// Image Filtering
NodeFactory.AddNodeAsPrototype('Vision/Image Filtering/F_VN_BilateralFilter', node_F_VN_BilateralFilter);
NodeFactory.AddNodeAsPrototype('Vision/Image Filtering/F_VN_BilateralFilterExp', node_F_VN_BilateralFilterExp);
NodeFactory.AddNodeAsPrototype('Vision/Image Filtering/F_VN_BoxFilter', node_F_VN_BoxFilter);
NodeFactory.AddNodeAsPrototype('Vision/Image Filtering/F_VN_BoxFilterExp', node_F_VN_BoxFilterExp);
NodeFactory.AddNodeAsPrototype('Vision/Image Filtering/F_VN_BrightBorderObjects', node_F_VN_BrightBorderObjects);
NodeFactory.AddNodeAsPrototype('Vision/Image Filtering/F_VN_CreateStructuringElement', node_F_VN_CreateStructuringElement);
//NodeFactory.AddNodeAsPrototype('Vision/Image Filtering/F_VN_CustomFilter', node_F_VN_CustomFilter);
//NodeFactory.AddNodeAsPrototype('Vision/Image Filtering/F_VN_CustomFilterExp', node_F_VN_CustomFilterExp);
NodeFactory.AddNodeAsPrototype('Vision/Image Filtering/F_VN_DarkBorderObjects', node_F_VN_DarkBorderObjects);
NodeFactory.AddNodeAsPrototype('Vision/Image Filtering/F_VN_FillHoles', node_F_VN_FillHoles);
NodeFactory.AddNodeAsPrototype('Vision/Image Filtering/F_VN_GaussianFilter', node_F_VN_GaussianFilter);
NodeFactory.AddNodeAsPrototype('Vision/Image Filtering/F_VN_GaussianFilterExp', node_F_VN_GaussianFilterExp);
NodeFactory.AddNodeAsPrototype('Vision/Image Filtering/F_VN_LaplacianFilter', node_F_VN_LaplacianFilter);
NodeFactory.AddNodeAsPrototype('Vision/Image Filtering/F_VN_LaplacianFilterExp', node_F_VN_LaplacianFilterExp);
NodeFactory.AddNodeAsPrototype('Vision/Image Filtering/F_VN_LocalMaxima', node_F_VN_LocalMaxima);
NodeFactory.AddNodeAsPrototype('Vision/Image Filtering/F_VN_LocalMinima', node_F_VN_LocalMinima);
NodeFactory.AddNodeAsPrototype('Vision/Image Filtering/F_VN_MedianFilter', node_F_VN_MedianFilter);
NodeFactory.AddNodeAsPrototype('Vision/Image Filtering/F_VN_MorphologicalOperator', node_F_VN_MorphologicalOperator);
NodeFactory.AddNodeAsPrototype('Vision/Image Filtering/F_VN_RemoveLocalMaxima', node_F_VN_RemoveLocalMaxima);
NodeFactory.AddNodeAsPrototype('Vision/Image Filtering/F_VN_RemoveLocalMinima', node_F_VN_RemoveLocalMinima);
NodeFactory.AddNodeAsPrototype('Vision/Image Filtering/F_VN_ScharrFilter', node_F_VN_ScharrFilter);
NodeFactory.AddNodeAsPrototype('Vision/Image Filtering/F_VN_ScharrFilterExp', node_F_VN_ScharrFilterExp);
//NodeFactory.AddNodeAsPrototype('Vision/Image Filtering/F_VN_SeparableCustomFilter', node_F_VN_SeparableCustomFilter);
//NodeFactory.AddNodeAsPrototype('Vision/Image Filtering/F_VN_SeparableCustomFilterExp', node_F_VN_SeparableCustomFilterExp);
NodeFactory.AddNodeAsPrototype('Vision/Image Filtering/F_VN_SobelFilter', node_F_VN_SobelFilter);
NodeFactory.AddNodeAsPrototype('Vision/Image Filtering/F_VN_SobelFilterExp', node_F_VN_SobelFilterExp);
NodeFactory.AddNodeAsPrototype('Vision/Image Filtering/F_VN_VarianceFilter', node_F_VN_VarianceFilter);
NodeFactory.AddNodeAsPrototype('Vision/Image Filtering/F_VN_VarianceFilterExp', node_F_VN_VarianceFilterExp);
    
// Image Segmentation
NodeFactory.AddNodeAsPrototype('Vision/Image Segmentation/F_VN_AdaptiveThreshold', node_F_VN_AdaptiveThreshold);
NodeFactory.AddNodeAsPrototype('Vision/Image Segmentation/F_VN_AdaptiveThresholdExp', node_F_VN_AdaptiveThresholdExp);
NodeFactory.AddNodeAsPrototype('Vision/Image Segmentation/F_VN_CheckColorRange', node_F_VN_CheckColorRange);
NodeFactory.AddNodeAsPrototype('Vision/Image Segmentation/F_VN_DoubleThreshold', node_F_VN_DoubleThreshold);
NodeFactory.AddNodeAsPrototype('Vision/Image Segmentation/F_VN_Threshold', node_F_VN_Threshold);
NodeFactory.AddNodeAsPrototype('Vision/Image Segmentation/F_VN_WatershedSegmentationExp', node_F_VN_WatershedSegmentationExp);
NodeFactory.AddNodeAsPrototype('Vision/Image Segmentation/F_VN_SauvolaThreshold', node_F_VN_SauvolaThreshold);

// Keypoint Features
NodeFactory.AddNodeAsPrototype('Vision/Keypoint Features/F_VN_FilterGoodMatches', node_F_VN_FilterGoodMatches);
NodeFactory.AddNodeAsPrototype('Vision/Keypoint Features/F_VN_FindReferenceKeyPointsInImage', node_F_VN_FindReferenceKeyPointsInImage);
NodeFactory.AddNodeAsPrototype('Vision/Keypoint Features/F_VN_FindReferenceKeyPointsInImageAKAZE', node_F_VN_FindReferenceKeyPointsInImageAKAZE);
NodeFactory.AddNodeAsPrototype('Vision/Keypoint Features/F_VN_FindReferenceKeyPointsInImageAKAZEExp', node_F_VN_FindReferenceKeyPointsInImageAKAZEExp);
NodeFactory.AddNodeAsPrototype('Vision/Keypoint Features/F_VN_FindReferenceKeyPointsInImageBRISK', node_F_VN_FindReferenceKeyPointsInImageBRISK);
NodeFactory.AddNodeAsPrototype('Vision/Keypoint Features/F_VN_FindReferenceKeyPointsInImageBRISKExp', node_F_VN_FindReferenceKeyPointsInImageBRISKExp);
NodeFactory.AddNodeAsPrototype('Vision/Keypoint Features/F_VN_FindReferenceKeyPointsInImageExp', node_F_VN_FindReferenceKeyPointsInImageExp);
NodeFactory.AddNodeAsPrototype('Vision/Keypoint Features/F_VN_FindReferenceKeyPointsInImageORB', node_F_VN_FindReferenceKeyPointsInImageORB);
NodeFactory.AddNodeAsPrototype('Vision/Keypoint Features/F_VN_FindReferenceKeyPointsInImageORBExp', node_F_VN_FindReferenceKeyPointsInImageORBExp);
NodeFactory.AddNodeAsPrototype('Vision/Keypoint Features/F_VN_GetMatchCoordinates', node_F_VN_GetMatchCoordinates);
NodeFactory.AddNodeAsPrototype('Vision/Keypoint Features/F_VN_KeyPointsAGAST', node_F_VN_KeyPointsAGAST);
NodeFactory.AddNodeAsPrototype('Vision/Keypoint Features/F_VN_KeyPointsAGASTExp', node_F_VN_KeyPointsAGASTExp);
NodeFactory.AddNodeAsPrototype('Vision/Keypoint Features/F_VN_KeyPointsAndDescriptorsAKAZE', node_F_VN_KeyPointsAndDescriptorsAKAZE);
NodeFactory.AddNodeAsPrototype('Vision/Keypoint Features/F_VN_KeyPointsAndDescriptorsAKAZEExp', node_F_VN_KeyPointsAndDescriptorsAKAZEExp);
NodeFactory.AddNodeAsPrototype('Vision/Keypoint Features/F_VN_KeyPointsAndDescriptorsBRISK', node_F_VN_KeyPointsAndDescriptorsBRISK);
NodeFactory.AddNodeAsPrototype('Vision/Keypoint Features/F_VN_KeyPointsAndDescriptorsBRISKExp', node_F_VN_KeyPointsAndDescriptorsBRISKExp);
NodeFactory.AddNodeAsPrototype('Vision/Keypoint Features/F_VN_KeyPointsAndDescriptorsKAZE', node_F_VN_KeyPointsAndDescriptorsKAZE);
NodeFactory.AddNodeAsPrototype('Vision/Keypoint Features/F_VN_KeyPointsAndDescriptorsKAZEExp', node_F_VN_KeyPointsAndDescriptorsKAZEExp);
NodeFactory.AddNodeAsPrototype('Vision/Keypoint Features/F_VN_KeyPointsAndDescriptorsORB', node_F_VN_KeyPointsAndDescriptorsORB);
NodeFactory.AddNodeAsPrototype('Vision/Keypoint Features/F_VN_KeyPointsAndDescriptorsORBExp', node_F_VN_KeyPointsAndDescriptorsORBExp);
NodeFactory.AddNodeAsPrototype('Vision/Keypoint Features/F_VN_KeyPointsFAST', node_F_VN_KeyPointsFAST);
NodeFactory.AddNodeAsPrototype('Vision/Keypoint Features/F_VN_KeyPointsFASTExp', node_F_VN_KeyPointsFASTExp);
NodeFactory.AddNodeAsPrototype('Vision/Keypoint Features/F_VN_KeyPointsGFTT', node_F_VN_KeyPointsGFTT);
NodeFactory.AddNodeAsPrototype('Vision/Keypoint Features/F_VN_KeyPointsGFTTExp', node_F_VN_KeyPointsGFTTExp);
NodeFactory.AddNodeAsPrototype('Vision/Keypoint Features/F_VN_KeyPointsMSER', node_F_VN_KeyPointsMSER);
NodeFactory.AddNodeAsPrototype('Vision/Keypoint Features/F_VN_KeyPointsMSERExp', node_F_VN_KeyPointsMSERExp);
NodeFactory.AddNodeAsPrototype('Vision/Keypoint Features/F_VN_KeyPointsSB', node_F_VN_KeyPointsSB);
NodeFactory.AddNodeAsPrototype('Vision/Keypoint Features/F_VN_KeyPointsSBExp', node_F_VN_KeyPointsSBExp);
NodeFactory.AddNodeAsPrototype('Vision/Keypoint Features/F_VN_MatchDescriptorsBF', node_F_VN_MatchDescriptorsBF);
NodeFactory.AddNodeAsPrototype('Vision/Keypoint Features/F_VN_MatchDescriptorsBFExp', node_F_VN_MatchDescriptorsBFExp);
NodeFactory.AddNodeAsPrototype('Vision/Keypoint Features/F_VN_MatchDescriptorsFlannLsh', node_F_VN_MatchDescriptorsFlannLsh);
NodeFactory.AddNodeAsPrototype('Vision/Keypoint Features/F_VN_MatchDescriptorsFlannLshExp', node_F_VN_MatchDescriptorsFlannLshExp);
NodeFactory.AddNodeAsPrototype('Vision/Keypoint Features/F_VN_MatchDescriptorsKnnBF', node_F_VN_MatchDescriptorsKnnBF);
NodeFactory.AddNodeAsPrototype('Vision/Keypoint Features/F_VN_MatchDescriptorsKnnBFExp', node_F_VN_MatchDescriptorsKnnBFExp);
NodeFactory.AddNodeAsPrototype('Vision/Keypoint Features/F_VN_MatchDescriptorsKnnFlannLsh', node_F_VN_MatchDescriptorsKnnFlannLsh);
NodeFactory.AddNodeAsPrototype('Vision/Keypoint Features/F_VN_MatchDescriptorsKnnFlannLshExp', node_F_VN_MatchDescriptorsKnnFlannLshExp);
NodeFactory.AddNodeAsPrototype('Vision/Keypoint Features/F_VN_RegionsMSER', node_F_VN_RegionsMSER);
NodeFactory.AddNodeAsPrototype('Vision/Keypoint Features/F_VN_RegionsMSERExp', node_F_VN_RegionsMSERExp);

// Machine Learning
//NodeFactory.AddNodeAsPrototype('Vision/Machine Learning/F_VN_CreateBoostClassifier', node_F_VN_CreateBoostClassifier);
//NodeFactory.AddNodeAsPrototype('Vision/Machine Learning/F_VN_CreateBoostClassifierExp', node_F_VN_CreateBoostClassifierExp);
//NodeFactory.AddNodeAsPrototype('Vision/Machine Learning/F_VN_CreateBoostClassifierExp2', node_F_VN_CreateBoostClassifierExp2);
//NodeFactory.AddNodeAsPrototype('Vision/Machine Learning/F_VN_CreateKmppModel', node_F_VN_CreateKmppModel);
//NodeFactory.AddNodeAsPrototype('Vision/Machine Learning/F_VN_CreateKmppModelExp', node_F_VN_CreateKmppModelExp);
//NodeFactory.AddNodeAsPrototype('Vision/Machine Learning/F_VN_CreateKnnModel', node_F_VN_CreateKnnModel);
//NodeFactory.AddNodeAsPrototype('Vision/Machine Learning/F_VN_CreateLbgModel', node_F_VN_CreateLbgModel);
//NodeFactory.AddNodeAsPrototype('Vision/Machine Learning/F_VN_CreateLbgModelExp', node_F_VN_CreateLbgModelExp);
//NodeFactory.AddNodeAsPrototype('Vision/Machine Learning/F_VN_CreateLdaTransform', node_F_VN_CreateLdaTransform);
//NodeFactory.AddNodeAsPrototype('Vision/Machine Learning/F_VN_CreateLdaTransformViaComponentNum', node_F_VN_CreateLdaTransformViaComponentNum);
//NodeFactory.AddNodeAsPrototype('Vision/Machine Learning/F_VN_CreateNbcModel', node_F_VN_CreateNbcModel);
//NodeFactory.AddNodeAsPrototype('Vision/Machine Learning/F_VN_CreatePcaTransform', node_F_VN_CreatePcaTransform);
//NodeFactory.AddNodeAsPrototype('Vision/Machine Learning/F_VN_CreatePcaTransformViaComponentNum', node_F_VN_CreatePcaTransformViaComponentNum);
//NodeFactory.AddNodeAsPrototype('Vision/Machine Learning/F_VN_CreatePcaTransformViaVariance', node_F_VN_CreatePcaTransformViaVariance);
//NodeFactory.AddNodeAsPrototype('Vision/Machine Learning/F_VN_CreateRTreesModel', node_F_VN_CreateRTreesModel);
//NodeFactory.AddNodeAsPrototype('Vision/Machine Learning/F_VN_CreateRTreesModelExp', node_F_VN_CreateRTreesModelExp);
//NodeFactory.AddNodeAsPrototype('Vision/Machine Learning/F_VN_CreateRTreesModelExp2', node_F_VN_CreateRTreesModelExp2);
//NodeFactory.AddNodeAsPrototype('Vision/Machine Learning/F_VN_CreateStaModel', node_F_VN_CreateStaModel);
//NodeFactory.AddNodeAsPrototype('Vision/Machine Learning/F_VN_CreateStaModelExp', node_F_VN_CreateStaModelExp);
//NodeFactory.AddNodeAsPrototype('Vision/Machine Learning/F_VN_CreateStaModelExp2', node_F_VN_CreateStaModelExp2);
//NodeFactory.AddNodeAsPrototype('Vision/Machine Learning/F_VN_CreateSvmModel', node_F_VN_CreateSvmModel);
//NodeFactory.AddNodeAsPrototype('Vision/Machine Learning/F_VN_CreateSvmModelExp', node_F_VN_CreateSvmModelExp);
//NodeFactory.AddNodeAsPrototype('Vision/Machine Learning/F_VN_CreateSvmModelExp2', node_F_VN_CreateSvmModelExp2);
//NodeFactory.AddNodeAsPrototype('Vision/Machine Learning/F_VN_CreateSvmSgdClassifier', node_F_VN_CreateSvmSgdClassifier);
//NodeFactory.AddNodeAsPrototype('Vision/Machine Learning/F_VN_CreateSvmSgdClassifierExp', node_F_VN_CreateSvmSgdClassifierExp);
//NodeFactory.AddNodeAsPrototype('Vision/Machine Learning/F_VN_FeatureScaling', node_F_VN_FeatureScaling);
//NodeFactory.AddNodeAsPrototype('Vision/Machine Learning/F_VN_FeatureScalingExp', node_F_VN_FeatureScalingExp);
//NodeFactory.AddNodeAsPrototype('Vision/Machine Learning/F_VN_FeatureTransform', node_F_VN_FeatureTransform);
//NodeFactory.AddNodeAsPrototype('Vision/Machine Learning/F_VN_GetBatchClusters', node_F_VN_GetBatchClusters);
//NodeFactory.AddNodeAsPrototype('Vision/Machine Learning/F_VN_GetBatchClustersExp', node_F_VN_GetBatchClustersExp);
//NodeFactory.AddNodeAsPrototype('Vision/Machine Learning/F_VN_GetBatchNovelties', node_F_VN_GetBatchNovelties);
//NodeFactory.AddNodeAsPrototype('Vision/Machine Learning/F_VN_GetClusterCenter', node_F_VN_GetClusterCenter);
//NodeFactory.AddNodeAsPrototype('Vision/Machine Learning/F_VN_GetClusterNum', node_F_VN_GetClusterNum);
//NodeFactory.AddNodeAsPrototype('Vision/Machine Learning/F_VN_GetFeatureScales', node_F_VN_GetFeatureScales);
//NodeFactory.AddNodeAsPrototype('Vision/Machine Learning/F_VN_GetSampleCluster', node_F_VN_GetSampleCluster);
//NodeFactory.AddNodeAsPrototype('Vision/Machine Learning/F_VN_GetSampleClusterExp', node_F_VN_GetSampleClusterExp);
//NodeFactory.AddNodeAsPrototype('Vision/Machine Learning/F_VN_GetSampleNovelty', node_F_VN_GetSampleNovelty);
//NodeFactory.AddNodeAsPrototype('Vision/Machine Learning/F_VN_InverseFeatureScaling', node_F_VN_InverseFeatureScaling);
//NodeFactory.AddNodeAsPrototype('Vision/Machine Learning/F_VN_InverseFeatureScaling_REAL', node_F_VN_InverseFeatureScaling_REAL);
//NodeFactory.AddNodeAsPrototype('Vision/Machine Learning/F_VN_InverseFeatureScalingExp', node_F_VN_InverseFeatureScalingExp);
//NodeFactory.AddNodeAsPrototype('Vision/Machine Learning/F_VN_InverseFeatureScalingExp_REAL', node_F_VN_InverseFeatureScalingExp_REAL);
//NodeFactory.AddNodeAsPrototype('Vision/Machine Learning/F_VN_InverseFeatureTransform', node_F_VN_InverseFeatureTransform);
//NodeFactory.AddNodeAsPrototype('Vision/Machine Learning/F_VN_PredictBatch', node_F_VN_PredictBatch);
//NodeFactory.AddNodeAsPrototype('Vision/Machine Learning/F_VN_PredictBatchExp', node_F_VN_PredictBatchExp);
//NodeFactory.AddNodeAsPrototype('Vision/Machine Learning/F_VN_PredictSampleClass', node_F_VN_PredictSampleClass);
//NodeFactory.AddNodeAsPrototype('Vision/Machine Learning/F_VN_PredictSampleClassExp', node_F_VN_PredictSampleClassExp);
//NodeFactory.AddNodeAsPrototype('Vision/Machine Learning/F_VN_PredictSampleScalar', node_F_VN_PredictSampleScalar);
//NodeFactory.AddNodeAsPrototype('Vision/Machine Learning/F_VN_PredictSampleScalarExp', node_F_VN_PredictSampleScalarExp);
//NodeFactory.AddNodeAsPrototype('Vision/Machine Learning/F_VN_PredictSampleVector', node_F_VN_PredictSampleVector);
//NodeFactory.AddNodeAsPrototype('Vision/Machine Learning/F_VN_PredictSampleVectorExp', node_F_VN_PredictSampleVectorExp);
//NodeFactory.AddNodeAsPrototype('Vision/Machine Learning/F_VN_TrainBatch', node_F_VN_TrainBatch);
//NodeFactory.AddNodeAsPrototype('Vision/Machine Learning/F_VN_TrainBatchClusters', node_F_VN_TrainBatchClusters);
//NodeFactory.AddNodeAsPrototype('Vision/Machine Learning/F_VN_TrainSample', node_F_VN_TrainSample);
//NodeFactory.AddNodeAsPrototype('Vision/Machine Learning/F_VN_TrainSampleClass', node_F_VN_TrainSampleClass);
//NodeFactory.AddNodeAsPrototype('Vision/Machine Learning/F_VN_TrainSampleCluster', node_F_VN_TrainSampleCluster);
//NodeFactory.AddNodeAsPrototype('Vision/Machine Learning/F_VN_TrainSampleScalar', node_F_VN_TrainSampleScalar
//NodeFactory.AddNodeAsPrototype('Vision/Machine Learning/F_VN_TrainSampleVector', node_F_VN_TrainSampleVector);

// Measurement
NodeFactory.AddNodeAsPrototype('Vision/Measurement/F_VN_AdjustSearchWindowOrientationToLinearEdge', node_F_VN_AdjustSearchWindowOrientationToLinearEdge);
NodeFactory.AddNodeAsPrototype('Vision/Measurement/F_VN_ClosestPointsBF', node_F_VN_ClosestPointsBF);
NodeFactory.AddNodeAsPrototype('Vision/Measurement/F_VN_LocateAxisAlignedEdges', node_F_VN_LocateAxisAlignedEdges);
NodeFactory.AddNodeAsPrototype('Vision/Measurement/F_VN_LocateAxisAlignedEdgesExp', node_F_VN_LocateAxisAlignedEdgesExp);
NodeFactory.AddNodeAsPrototype('Vision/Measurement/F_VN_LocateCircularArc', node_F_VN_LocateCircularArc);
NodeFactory.AddNodeAsPrototype('Vision/Measurement/F_VN_LocateCircularArcExp', node_F_VN_LocateCircularArcExp);
NodeFactory.AddNodeAsPrototype('Vision/Measurement/F_VN_LocateCircularArcExp2', node_F_VN_LocateCircularArcExp2);
NodeFactory.AddNodeAsPrototype('Vision/Measurement/F_VN_LocateEdge', node_F_VN_LocateEdge);
NodeFactory.AddNodeAsPrototype('Vision/Measurement/F_VN_LocateEdgeExp', node_F_VN_LocateEdgeExp);
NodeFactory.AddNodeAsPrototype('Vision/Measurement/F_VN_LocateEdgeExp2', node_F_VN_LocateEdgeExp2);
NodeFactory.AddNodeAsPrototype('Vision/Measurement/F_VN_LocateEdges', node_F_VN_LocateEdges);
NodeFactory.AddNodeAsPrototype('Vision/Measurement/F_VN_LocateEdgesExp', node_F_VN_LocateEdgesExp);
NodeFactory.AddNodeAsPrototype('Vision/Measurement/F_VN_LocateEdgesExp2', node_F_VN_LocateEdgesExp2);
NodeFactory.AddNodeAsPrototype('Vision/Measurement/F_VN_LocateEllipse', node_F_VN_LocateEllipse);
NodeFactory.AddNodeAsPrototype('Vision/Measurement/F_VN_LocateEllipseExp', node_F_VN_LocateEllipseExp);
NodeFactory.AddNodeAsPrototype('Vision/Measurement/F_VN_LocateEllipseExp2', node_F_VN_LocateEllipseExp2);
NodeFactory.AddNodeAsPrototype('Vision/Measurement/F_VN_MeasureAngleBetweenEdges', node_F_VN_MeasureAngleBetweenEdges);
NodeFactory.AddNodeAsPrototype('Vision/Measurement/F_VN_MeasureAngleBetweenEdgesExp', node_F_VN_MeasureAngleBetweenEdgesExp);
NodeFactory.AddNodeAsPrototype('Vision/Measurement/F_VN_MeasureAngleBetweenEdgesExp2', node_F_VN_MeasureAngleBetweenEdgesExp2);
NodeFactory.AddNodeAsPrototype('Vision/Measurement/F_VN_MeasureEdgeDistance', node_F_VN_MeasureEdgeDistance);
NodeFactory.AddNodeAsPrototype('Vision/Measurement/F_VN_MeasureEdgeDistanceExp', node_F_VN_MeasureEdgeDistanceExp);
NodeFactory.AddNodeAsPrototype('Vision/Measurement/F_VN_MeasureEdgeDistanceExp2', node_F_VN_MeasureEdgeDistanceExp2);
NodeFactory.AddNodeAsPrototype('Vision/Measurement/F_VN_MeasureMinEdgeDistance', node_F_VN_MeasureMinEdgeDistance);
NodeFactory.AddNodeAsPrototype('Vision/Measurement/F_VN_MeasureMinEdgeDistanceExp', node_F_VN_MeasureMinEdgeDistanceExp);
NodeFactory.AddNodeAsPrototype('Vision/Measurement/F_VN_MeasureMinEdgeDistanceExp2', node_F_VN_MeasureMinEdgeDistanceExp2);

// Miscellaneous
NodeFactory.AddNodeAsPrototype('Vision/Miscellaneous/F_VN_CheckFunctionInitialization', node_F_VN_CheckFunctionInitialization);
NodeFactory.AddNodeAsPrototype('Vision/Miscellaneous/F_VN_ClipLineToBoundary', node_F_VN_ClipLineToBoundary);
NodeFactory.AddNodeAsPrototype('Vision/Miscellaneous/F_VN_ClipLineToBoundary_ITcVnImage', node_F_VN_ClipLineToBoundary_ITcVnImage);
NodeFactory.AddNodeAsPrototype('Vision/Miscellaneous/F_VN_ClipLineToBoundary_TcVnRectangle_DINT', node_F_VN_ClipLineToBoundary_TcVnRectangle_DINT);
//NodeFactory.AddNodeAsPrototype('Vision/Miscellaneous/F_VN_ConvertITcUnknownToITcVnBitmapExport', node_F_VN_ConvertITcUnknownToITcVnBitmapExport);
//NodeFactory.AddNodeAsPrototype('Vision/Miscellaneous/F_VN_ConvertITcUnknownToITcVnContainer', node_F_VN_ConvertITcUnknownToITcVnContainer);
//NodeFactory.AddNodeAsPrototype('Vision/Miscellaneous/F_VN_ConvertITcUnknownToITcVnImage', node_F_VN_ConvertITcUnknownToITcVnImage);
//NodeFactory.AddNodeAsPrototype('Vision/Miscellaneous/F_VN_ConvertITcUnknownToITcVnMlModel', node_F_VN_ConvertITcUnknownToITcVnMlModel);
NodeFactory.AddNodeAsPrototype('Vision/Miscellaneous/F_VN_DeinitializeFunction', node_F_VN_DeinitializeFunction);
//NodeFactory.AddNodeAsPrototype('Vision/Miscellaneous/F_VN_GetTimestamp', node_F_VN_GetTimestamp);
NodeFactory.AddNodeAsPrototype('Vision/Miscellaneous/F_VN_HuMomentInvariants', node_F_VN_HuMomentInvariants);
//NodeFactory.AddNodeAsPrototype('Vision/Miscellaneous/F_VN_InitMatrixStruct', node_F_VN_InitMatrixStruct);
NodeFactory.AddNodeAsPrototype('Vision/Miscellaneous/F_VN_InvertMatrix3x3', node_F_VN_InvertMatrix3x3);
NodeFactory.AddNodeAsPrototype('Vision/Miscellaneous/F_VN_LineIntersectionPoint', node_F_VN_LineIntersectionPoint);
NodeFactory.AddNodeAsPrototype('Vision/Miscellaneous/F_VN_LineIntersectionPointAndAngle', node_F_VN_LineIntersectionPointAndAngle);
//NodeFactory.AddNodeAsPrototype('Vision/Miscellaneous/F_VN_MultiplyMatrices', node_F_VN_MultiplyMatrices);
NodeFactory.AddNodeAsPrototype('Vision/Miscellaneous/F_VN_OrthogonalVector_TcVnVector2_DINT', node_F_VN_OrthogonalVector_TcVnVector2_DINT);
NodeFactory.AddNodeAsPrototype('Vision/Miscellaneous/F_VN_OrthogonalVector_TcVnVector2_LREAL', node_F_VN_OrthogonalVector_TcVnVector2_LREAL);
NodeFactory.AddNodeAsPrototype('Vision/Miscellaneous/F_VN_OrthogonalVector_TcVnVector2_REAL', node_F_VN_OrthogonalVector_TcVnVector2_REAL);
NodeFactory.AddNodeAsPrototype('Vision/Miscellaneous/F_VN_PointToLineDistance_TcVnPoint2_DINT', node_F_VN_PointToLineDistance_TcVnPoint2_DINT);
NodeFactory.AddNodeAsPrototype('Vision/Miscellaneous/F_VN_PointToLineDistance_TcVnPoint2_LREAL', node_F_VN_PointToLineDistance_TcVnPoint2_LREAL);
NodeFactory.AddNodeAsPrototype('Vision/Miscellaneous/F_VN_PointToLineDistance_TcVnPoint2_REAL', node_F_VN_PointToLineDistance_TcVnPoint2_REAL);
NodeFactory.AddNodeAsPrototype('Vision/Miscellaneous/F_VN_PointToPointDirection_TcVnPoint2_DINT', node_F_VN_PointToPointDirection_TcVnPoint2_DINT);
NodeFactory.AddNodeAsPrototype('Vision/Miscellaneous/F_VN_PointToPointDirection_TcVnPoint2_LREAL', node_F_VN_PointToPointDirection_TcVnPoint2_LREAL);
NodeFactory.AddNodeAsPrototype('Vision/Miscellaneous/F_VN_PointToPointDirection_TcVnPoint2_REAL', node_F_VN_PointToPointDirection_TcVnPoint2_REAL);
NodeFactory.AddNodeAsPrototype('Vision/Miscellaneous/F_VN_PointToPointDistance_TcVnPoint2_DINT', node_F_VN_PointToPointDistance_TcVnPoint2_DINT);
NodeFactory.AddNodeAsPrototype('Vision/Miscellaneous/F_VN_PointToPointDistance_TcVnPoint2_LREAL', node_F_VN_PointToPointDistance_TcVnPoint2_LREAL);
NodeFactory.AddNodeAsPrototype('Vision/Miscellaneous/F_VN_PointToPointDistance_TcVnPoint2_REAL', node_F_VN_PointToPointDistance_TcVnPoint2_REAL);
NodeFactory.AddNodeAsPrototype('Vision/Miscellaneous/F_VN_RotatedRectangleCorners', node_F_VN_RotatedRectangleCorners);
NodeFactory.AddNodeAsPrototype('Vision/Miscellaneous/F_VN_RotatedRectangleIntersection', node_F_VN_RotatedRectangleIntersection);
//NodeFactory.AddNodeAsPrototype('Vision/Miscellaneous/F_VN_SetRngSeed', node_F_VN_SetRngSeed);
//NodeFactory.AddNodeAsPrototype('Vision/Miscellaneous/F_VN_UpdateTimestamp', node_F_VN_UpdateTimestamp);

// NodeFactory.AddNodeAsPrototype('Vision/Miscellaneous/FB_VN_InitializeFunction', node_FB_VN_InitializeFunction);

// OCR
NodeFactory.AddNodeAsPrototype('Vision/OCR/F_VN_OCR', node_F_VN_OCR);
NodeFactory.AddNodeAsPrototype('Vision/OCR/F_VN_OCRExp', node_F_VN_OCRExp);

// Texture Analysis
NodeFactory.AddNodeAsPrototype('Vision/Texture Analysis/F_VN_Granulometry', node_F_VN_Granulometry);
NodeFactory.AddNodeAsPrototype('Vision/Texture Analysis/F_VN_HaralickFeatures', node_F_VN_HaralickFeatures);

// Neural Network
//NodeFactory.AddNodeAsPrototype('Vision/Neural Network/F_VN_ConvertDataLayout', node_F_VN_ConvertDataLayout);
//NodeFactory.AddNodeAsPrototype('Vision/Neural Network/F_VN_ExecuteNeuralNetwork', node_F_VN_ExecuteNeuralNetwork);
//NodeFactory.AddNodeAsPrototype('Vision/Neural Network/F_VN_ExecuteNeuralNetwork_MultiLayerOutput', node_F_VN_ExecuteNeuralNetwork_MultiLayerOutput);
//NodeFactory.AddNodeAsPrototype('Vision/Neural Network/F_VN_ExecuteNeuralNetwork_SingleLayerOutput', node_F_VN_ExecuteNeuralNetwork_SingleLayerOutput);
//NodeFactory.AddNodeAsPrototype('Vision/Neural Network/F_VN_GetNeuralNetworkLayerNames', node_F_VN_GetNeuralNetworkLayerNames);
//NodeFactory.AddNodeAsPrototype('Vision/Neural Network/F_VN_NonMaxSuppression', node_F_VN_NonMaxSuppression);
//NodeFactory.AddNodeAsPrototype('Vision/Neural Network/F_VN_NonMaxSuppressionExp', node_F_VN_NonMaxSuppressionExp);
NodeFactory.AddNodeAsPrototype('Vision/Neural Network/F_VN_Reduce', node_F_VN_Reduce);
NodeFactory.AddNodeAsPrototype('Vision/Neural Network/F_VN_ReduceArg', node_F_VN_ReduceArg);
//NodeFactory.AddNodeAsPrototype('Vision/Neural Network/F_VN_ReshapeImage', node_F_VN_ReshapeImage);
NodeFactory.AddNodeAsPrototype('Vision/Neural Network/F_VN_Sigmoid', node_F_VN_Sigmoid);
NodeFactory.AddNodeAsPrototype('Vision/Neural Network/F_VN_SigmoidExp', node_F_VN_SigmoidExp);
NodeFactory.AddNodeAsPrototype('Vision/Neural Network/F_VN_SoftMax', node_F_VN_SoftMax);
END_METHOD

END_FUNCTION_BLOCK

// ---- Nodes/Contour Analysis/Node_F_VN_MatchContours.TcPOU
{attribute 'linkalways'}
{attribute 'no_explicit_call' := 'This FB is a CLASS and must be accessed using methods or properties'}
{attribute 'enable_dynamic_creation'}
FUNCTION_BLOCK Node_F_VN_MatchContours EXTENDS VisionNode
VAR
    ipContour1 : _ITcVnContainer;
    ipContour2 : _ITcVnContainer;
    eComparisonMethod : _ETcVnContoursMatchComparisonMethod(ETcVnContoursMatchComparisonMethod.TCVN_CMCM_CONTOURS_MATCH_I1);
    fDissimilarity : _LREAL(0.0);
    hrPrev : _HRESULT(S_OK);
    hresult : _HRESULT(S_OK);
END_VAR

METHOD PUBLIC Clone : I_Node
VAR
    pNode : POINTER TO Node_F_VN_MatchContours;
END_VAR
pNode := __NEW(Node_F_VN_MatchContours);
Clone := pNode^;
END_METHOD

METHOD FB_init : BOOL
VAR_INPUT
    bInitRetains : BOOL;
    bInCopyCode : BOOL;
END_VAR
AddInput('ipContour1', ipContour1);
AddInput('ipContour2', ipContour2);
AddParameter('eComparisonMethod', eComparisonMethod);
AddOutput('fDissimilarity', fDissimilarity);
AddInput('hrPrev', hrPrev);
AddOutput('hresult', hresult);
END_METHOD

METHOD PROTECTED OnExecute
hresult.Value := F_VN_MatchContours(
    ipContour1 := ipContour1.Value,
    ipContour2 := ipContour2.Value,
    eComparisonMethod := eComparisonMethod.Value,
    fDissimilarity := fDissimilarity.Value,
    hrPrev := hrPrev.Value);
END_METHOD

METHOD PUBLIC PreExecutionCheck
VAR_INPUT
    Check : I_PreExecutionChecks;
END_VAR
Check.IsTrue(ipContour1.IsValid, 'ipContour1 must contain a container');
Check.IsTrue(ipContour2.IsValid, 'ipContour2 must contain a container');
Check.IsTrue(ipContour1.IsType(TC_GLOBAL_CONST_LIST.ContainerType_Vector_TcVnPoint2_DINT) OR
             ipContour1.IsType(TC_GLOBAL_CONST_LIST.ContainerType_Vector_TcVnPoint2_REAL) OR
             ipContour1.IsType(TC_GLOBAL_CONST_LIST.ContainerType_Vector_Vector_TcVnPoint2_DINT), 'Unsupported contour container type');
Check.IsTrue(ContainersHaveMatchingTypes(ipContour1.Value, ipContour2.Value), 'Contours must have matching container types');
Check.IsTrue((eComparisonMethod.Value = ETcVnContoursMatchComparisonMethod.TCVN_CMCM_CONTOURS_MATCH_I1) OR
             (eComparisonMethod.Value = ETcVnContoursMatchComparisonMethod.TCVN_CMCM_CONTOURS_MATCH_I2) OR
             (eComparisonMethod.Value = ETcVnContoursMatchComparisonMethod.TCVN_CMCM_CONTOURS_MATCH_I3), 'Unsupported eComparisonMethod');
END_METHOD

END_FUNCTION_BLOCK

// ---- Nodes/Contour Analysis/Node_F_VN_MatchContoursExp.TcPOU
{attribute 'linkalways'}
{attribute 'no_explicit_call' := 'This FB is a CLASS and must be accessed using methods or properties'}
{attribute 'enable_dynamic_creation'}
FUNCTION_BLOCK Node_F_VN_MatchContoursExp EXTENDS VisionNode
VAR
    ipContour1 : _ITcVnContainer;
    ipContour2 : _ITcVnContainer;
    eComparisonMethod : _ETcVnContoursMatchComparisonMethod(ETcVnContoursMatchComparisonMethod.TCVN_CMCM_CONTOURS_MATCH_I1);
    fDissimilarity : _LREAL(0.0);
    fAreaFactor : _LREAL(0);
    fAbsPositionFactor : _LREAL(0);
    fRelPositionFactor : _LREAL(0);
    fNumDiffFactor : _LREAL(0);
    hrPrev : _HRESULT(S_OK);
    hresult : _HRESULT(S_OK);
END_VAR

METHOD PUBLIC Clone : I_Node
VAR
    pNode : POINTER TO Node_F_VN_MatchContoursExp;
END_VAR
pNode := __NEW(Node_F_VN_MatchContoursExp);
Clone := pNode^;
END_METHOD

METHOD FB_init : BOOL
VAR_INPUT
    bInitRetains : BOOL;
    bInCopyCode : BOOL;
END_VAR
AddInput('ipContour1', ipContour1);
AddInput('ipContour2', ipContour2);
AddParameter('eComparisonMethod', eComparisonMethod);
AddOutput('fDissimilarity', fDissimilarity);
AddParameter('fAreaFactor', fAreaFactor);
AddParameter('fAbsPositionFactor', fAbsPositionFactor);
AddParameter('fRelPositionFactor', fRelPositionFactor);
AddParameter('fNumDiffFactor', fNumDiffFactor);
AddInput('hrPrev', hrPrev);
AddOutput('hresult', hresult);
END_METHOD

METHOD PROTECTED OnExecute
hresult.Value := F_VN_MatchContoursExp(
    ipContour1 := ipContour1.Value,
    ipContour2 := ipContour2.Value,
    eComparisonMethod := eComparisonMethod.Value,
    fDissimilarity := fDissimilarity.Value,
    fAreaFactor := fAreaFactor.Value,
    fAbsPositionFactor := fAbsPositionFactor.Value,
    fRelPositionFactor := fRelPositionFactor.Value,
    fNumDiffFactor := fNumDiffFactor.Value,
    hrPrev := hrPrev.Value);
END_METHOD

METHOD PUBLIC PreExecutionCheck
VAR_INPUT
    Check : I_PreExecutionChecks;
END_VAR
Check.IsTrue(ipContour1.IsValid, 'ipContour1 must contain a container');
Check.IsTrue(ipContour2.IsValid, 'ipContour2 must contain a container');
Check.IsTrue(ipContour1.IsType(TC_GLOBAL_CONST_LIST.ContainerType_Vector_TcVnPoint2_DINT) OR
             ipContour1.IsType(TC_GLOBAL_CONST_LIST.ContainerType_Vector_TcVnPoint2_REAL) OR
             ipContour1.IsType(TC_GLOBAL_CONST_LIST.ContainerType_Vector_Vector_TcVnPoint2_DINT), 'Unsupported contour container type');
Check.IsTrue(ContainersHaveMatchingTypes(ipContour1.Value, ipContour2.Value), 'Contours must have matching container types');
Check.IsTrue((eComparisonMethod.Value = ETcVnContoursMatchComparisonMethod.TCVN_CMCM_CONTOURS_MATCH_I1) OR
             (eComparisonMethod.Value = ETcVnContoursMatchComparisonMethod.TCVN_CMCM_CONTOURS_MATCH_I2) OR
             (eComparisonMethod.Value = ETcVnContoursMatchComparisonMethod.TCVN_CMCM_CONTOURS_MATCH_I3), 'Unsupported eComparisonMethod');
END_METHOD

END_FUNCTION_BLOCK

// ---- Nodes/Geometric and Coord Transform/Node_F_VN_AlignRotatedImageRegionExp.TcPOU
{attribute 'linkalways'}
{attribute 'no_explicit_call' := 'This FB is a CLASS and must be accessed using methods or properties'}
{attribute 'enable_dynamic_creation'}
FUNCTION_BLOCK Node_F_VN_AlignRotatedImageRegionExp EXTENDS VisionNode
VAR
    ipSrcImage : _ITcVnImage;
    ipDestImage : _ITcVnImage;
    stRegion : _TcVnRotatedRectangle;
    eInterpolationType : _ETcVnInterpolationType(ETcVnInterpolationType.TCVN_IT_BILINEAR);
    eBorderInterpolation : _ETcVnBorderInterpolationMethod(ETcVnBorderInterpolationMethod.TCVN_BIM_CONSTANT);
    aBorderValue : _TcVnVector4_LREAL;
    hrPrev : _HRESULT(S_OK);
    hresult : _HRESULT(S_OK);
END_VAR

METHOD PUBLIC Clone : I_Node
VAR
    pNode : POINTER TO Node_F_VN_AlignRotatedImageRegionExp;
END_VAR
pNode := __NEW(Node_F_VN_AlignRotatedImageRegionExp);
Clone := pNode^;
END_METHOD

METHOD FB_init : BOOL
VAR_INPUT
    bInitRetains : BOOL;
    bInCopyCode : BOOL;
END_VAR
AddInput('ipSrcImage', ipSrcImage);
AddOutput('ipDestImage', ipDestImage);
AddInput('stRegion', stRegion);
AddParameter('eInterpolationType', eInterpolationType);
AddParameter('eBorderInterpolation', eBorderInterpolation);
AddInput('aBorderValue', aBorderValue);
AddInput('hrPrev', hrPrev);
AddOutput('hresult', hresult);
END_METHOD

METHOD PROTECTED OnExecute
hresult.Value := F_VN_AlignRotatedImageRegionExp(
    ipSrcImage := ipSrcImage.Value,
    ipDestImage := ipDestImage.Value,
    stRegion := stRegion.Value,
    eInterpolationType := eInterpolationType.Value,
    eBorderInterpolation := eBorderInterpolation.Value,
    aBorderValue := aBorderValue.Value,
    hrPrev := hrPrev.Value);
END_METHOD

METHOD PUBLIC PreExecutionCheck
VAR_INPUT
    Check : I_PreExecutionChecks;
END_VAR
Check.IsTrue(ipSrcImage.IsValid, 'ipSrcImage must contain an image');
Check.IsTrue(stRegion.Value.stSize.fWidth > 0.0, 'Region width must be positive');
Check.IsTrue(stRegion.Value.stSize.fHeight > 0.0, 'Region height must be positive');
Check.IsTrue((eInterpolationType.Value = ETcVnInterpolationType.TCVN_IT_NEAREST_NEIGHBOR) OR
             (eInterpolationType.Value = ETcVnInterpolationType.TCVN_IT_BILINEAR) OR
             (eInterpolationType.Value = ETcVnInterpolationType.TCVN_IT_BICUBIC) OR
             (eInterpolationType.Value = ETcVnInterpolationType.TCVN_IT_AREA_BASED) OR
             (eInterpolationType.Value = ETcVnInterpolationType.TCVN_IT_LANCZOS4), 'Unsupported eInterpolationType');
Check.IsTrue((eBorderInterpolation.Value = ETcVnBorderInterpolationMethod.TCVN_BIM_CONSTANT) OR
             (eBorderInterpolation.Value = ETcVnBorderInterpolationMethod.TCVN_BIM_REPLICATE) OR
             (eBorderInterpolation.Value = ETcVnBorderInterpolationMethod.TCVN_BIM_REFLECT) OR
             (eBorderInterpolation.Value = ETcVnBorderInterpolationMethod.TCVN_BIM_WRAP) OR
             (eBorderInterpolation.Value = ETcVnBorderInterpolationMethod.TCVN_BIM_REFLECT_101) OR
             (eBorderInterpolation.Value = ETcVnBorderInterpolationMethod.TCVN_BIM_DEFAULT) OR
             (eBorderInterpolation.Value = ETcVnBorderInterpolationMethod.TCVN_BIM_TRANSPARENT), 'Unsupported eBorderInterpolation');
END_METHOD

END_FUNCTION_BLOCK

// ---- Nodes/Geometric and Coord Transform/Node_F_VN_ConvertCartesianToPolarAngleImage.TcPOU
{attribute 'linkalways'}
{attribute 'no_explicit_call' := 'This FB is a CLASS and must be accessed using methods or properties'}
{attribute 'enable_dynamic_creation'}
FUNCTION_BLOCK Node_F_VN_ConvertCartesianToPolarAngleImage EXTENDS VisionNode
VAR
    ipSrcImageX : _ITcVnImage;
    ipSrcImageY : _ITcVnImage;
    ipDestImageAng : _ITcVnImage;
    hrPrev : _HRESULT(S_OK);
    hresult : _HRESULT(S_OK);
END_VAR

METHOD PUBLIC Clone : I_Node
VAR
    pNode : POINTER TO Node_F_VN_ConvertCartesianToPolarAngleImage;
END_VAR
pNode := __NEW(Node_F_VN_ConvertCartesianToPolarAngleImage);
Clone := pNode^;
END_METHOD

METHOD FB_init : BOOL
VAR_INPUT
    bInitRetains : BOOL;
    bInCopyCode : BOOL;
END_VAR
AddInput('ipSrcImageX', ipSrcImageX);
AddInput('ipSrcImageY', ipSrcImageY);
AddOutput('ipDestImageAng', ipDestImageAng);
AddInput('hrPrev', hrPrev);
AddOutput('hresult', hresult);
END_METHOD

METHOD PROTECTED OnExecute
hresult.Value := F_VN_ConvertCartesianToPolarAngleImage(
    ipSrcImageX := ipSrcImageX.Value,
    ipSrcImageY := ipSrcImageY.Value,
    ipDestImageAng := ipDestImageAng.Value,
    hrPrev := hrPrev.Value);
END_METHOD

METHOD PUBLIC PreExecutionCheck
VAR_INPUT
    Check : I_PreExecutionChecks;
END_VAR
Check.IsTrue(ipSrcImageX.IsValid, 'ipSrcImageX must contain an image');
Check.IsTrue(ipSrcImageX.IsElementType(ETcVnElementType.TCVN_ET_REAL) OR
             ipSrcImageX.IsElementType(ETcVnElementType.TCVN_ET_LREAL), 'Coordinate images must contain REAL or LREAL elements');
Check.IsTrue(ipSrcImageY.IsValid, 'ipSrcImageY must contain an image');
Check.IsTrue(ImagesHaveMatchingPixelFormats(ipSrcImageX.Value, ipSrcImageY.Value), 'Source images must have matching pixel formats');
Check.IsTrue(IsImage1SizeEqualToImage2Size(ipSrcImageX.Value, ipSrcImageY.Value), 'Source images must have matching dimensions');
END_METHOD

END_FUNCTION_BLOCK

// ---- Nodes/Geometric and Coord Transform/Node_F_VN_ConvertCartesianToPolarAngleImageExp.TcPOU
{attribute 'linkalways'}
{attribute 'no_explicit_call' := 'This FB is a CLASS and must be accessed using methods or properties'}
{attribute 'enable_dynamic_creation'}
FUNCTION_BLOCK Node_F_VN_ConvertCartesianToPolarAngleImageExp EXTENDS VisionNode
VAR
    ipSrcImageX : _ITcVnImage;
    ipSrcImageY : _ITcVnImage;
    ipDestImageAng : _ITcVnImage;
    bAngleInDegrees : _BOOL(FALSE);
    hrPrev : _HRESULT(S_OK);
    hresult : _HRESULT(S_OK);
END_VAR

METHOD PUBLIC Clone : I_Node
VAR
    pNode : POINTER TO Node_F_VN_ConvertCartesianToPolarAngleImageExp;
END_VAR
pNode := __NEW(Node_F_VN_ConvertCartesianToPolarAngleImageExp);
Clone := pNode^;
END_METHOD

METHOD FB_init : BOOL
VAR_INPUT
    bInitRetains : BOOL;
    bInCopyCode : BOOL;
END_VAR
AddInput('ipSrcImageX', ipSrcImageX);
AddInput('ipSrcImageY', ipSrcImageY);
AddOutput('ipDestImageAng', ipDestImageAng);
AddParameter('bAngleInDegrees', bAngleInDegrees);
AddInput('hrPrev', hrPrev);
AddOutput('hresult', hresult);
END_METHOD

METHOD PROTECTED OnExecute
hresult.Value := F_VN_ConvertCartesianToPolarAngleImageExp(
    ipSrcImageX := ipSrcImageX.Value,
    ipSrcImageY := ipSrcImageY.Value,
    ipDestImageAng := ipDestImageAng.Value,
    bAngleInDegrees := bAngleInDegrees.Value,
    hrPrev := hrPrev.Value);
END_METHOD

METHOD PUBLIC PreExecutionCheck
VAR_INPUT
    Check : I_PreExecutionChecks;
END_VAR
Check.IsTrue(ipSrcImageX.IsValid, 'ipSrcImageX must contain an image');
Check.IsTrue(ipSrcImageX.IsElementType(ETcVnElementType.TCVN_ET_REAL) OR
             ipSrcImageX.IsElementType(ETcVnElementType.TCVN_ET_LREAL), 'Coordinate images must contain REAL or LREAL elements');
Check.IsTrue(ipSrcImageY.IsValid, 'ipSrcImageY must contain an image');
Check.IsTrue(ImagesHaveMatchingPixelFormats(ipSrcImageX.Value, ipSrcImageY.Value), 'Source images must have matching pixel formats');
Check.IsTrue(IsImage1SizeEqualToImage2Size(ipSrcImageX.Value, ipSrcImageY.Value), 'Source images must have matching dimensions');
END_METHOD

END_FUNCTION_BLOCK

// ---- Nodes/Geometric and Coord Transform/Node_F_VN_ConvertCartesianToPolarImages.TcPOU
{attribute 'linkalways'}
{attribute 'no_explicit_call' := 'This FB is a CLASS and must be accessed using methods or properties'}
{attribute 'enable_dynamic_creation'}
FUNCTION_BLOCK Node_F_VN_ConvertCartesianToPolarImages EXTENDS VisionNode
VAR
    ipSrcImageX : _ITcVnImage;
    ipSrcImageY : _ITcVnImage;
    ipDestImageMag : _ITcVnImage;
    ipDestImageAng : _ITcVnImage;
    hrPrev : _HRESULT(S_OK);
    hresult : _HRESULT(S_OK);
END_VAR

METHOD PUBLIC Clone : I_Node
VAR
    pNode : POINTER TO Node_F_VN_ConvertCartesianToPolarImages;
END_VAR
pNode := __NEW(Node_F_VN_ConvertCartesianToPolarImages);
Clone := pNode^;
END_METHOD

METHOD FB_init : BOOL
VAR_INPUT
    bInitRetains : BOOL;
    bInCopyCode : BOOL;
END_VAR
AddInput('ipSrcImageX', ipSrcImageX);
AddInput('ipSrcImageY', ipSrcImageY);
AddOutput('ipDestImageMag', ipDestImageMag);
AddOutput('ipDestImageAng', ipDestImageAng);
AddInput('hrPrev', hrPrev);
AddOutput('hresult', hresult);
END_METHOD

METHOD PROTECTED OnExecute
hresult.Value := F_VN_ConvertCartesianToPolarImages(
    ipSrcImageX := ipSrcImageX.Value,
    ipSrcImageY := ipSrcImageY.Value,
    ipDestImageMag := ipDestImageMag.Value,
    ipDestImageAng := ipDestImageAng.Value,
    hrPrev := hrPrev.Value);
END_METHOD

METHOD PUBLIC PreExecutionCheck
VAR_INPUT
    Check : I_PreExecutionChecks;
END_VAR
Check.IsTrue(ipSrcImageX.IsValid, 'ipSrcImageX must contain an image');
Check.IsTrue(ipSrcImageX.IsElementType(ETcVnElementType.TCVN_ET_REAL) OR
             ipSrcImageX.IsElementType(ETcVnElementType.TCVN_ET_LREAL), 'Coordinate images must contain REAL or LREAL elements');
Check.IsTrue(ipSrcImageY.IsValid, 'ipSrcImageY must contain an image');
Check.IsTrue(ImagesHaveMatchingPixelFormats(ipSrcImageX.Value, ipSrcImageY.Value), 'Source images must have matching pixel formats');
Check.IsTrue(IsImage1SizeEqualToImage2Size(ipSrcImageX.Value, ipSrcImageY.Value), 'Source images must have matching dimensions');
END_METHOD

END_FUNCTION_BLOCK

// ---- Nodes/Geometric and Coord Transform/Node_F_VN_ConvertCartesianToPolarImagesExp.TcPOU
{attribute 'linkalways'}
{attribute 'no_explicit_call' := 'This FB is a CLASS and must be accessed using methods or properties'}
{attribute 'enable_dynamic_creation'}
FUNCTION_BLOCK Node_F_VN_ConvertCartesianToPolarImagesExp EXTENDS VisionNode
VAR
    ipSrcImageX : _ITcVnImage;
    ipSrcImageY : _ITcVnImage;
    ipDestImageMag : _ITcVnImage;
    ipDestImageAng : _ITcVnImage;
    bAngleInDegrees : _BOOL(FALSE);
    hrPrev : _HRESULT(S_OK);
    hresult : _HRESULT(S_OK);
END_VAR

METHOD PUBLIC Clone : I_Node
VAR
    pNode : POINTER TO Node_F_VN_ConvertCartesianToPolarImagesExp;
END_VAR
pNode := __NEW(Node_F_VN_ConvertCartesianToPolarImagesExp);
Clone := pNode^;
END_METHOD

METHOD FB_init : BOOL
VAR_INPUT
    bInitRetains : BOOL;
    bInCopyCode : BOOL;
END_VAR
AddInput('ipSrcImageX', ipSrcImageX);
AddInput('ipSrcImageY', ipSrcImageY);
AddOutput('ipDestImageMag', ipDestImageMag);
AddOutput('ipDestImageAng', ipDestImageAng);
AddParameter('bAngleInDegrees', bAngleInDegrees);
AddInput('hrPrev', hrPrev);
AddOutput('hresult', hresult);
END_METHOD

METHOD PROTECTED OnExecute
hresult.Value := F_VN_ConvertCartesianToPolarImagesExp(
    ipSrcImageX := ipSrcImageX.Value,
    ipSrcImageY := ipSrcImageY.Value,
    ipDestImageMag := ipDestImageMag.Value,
    ipDestImageAng := ipDestImageAng.Value,
    bAngleInDegrees := bAngleInDegrees.Value,
    hrPrev := hrPrev.Value);
END_METHOD

METHOD PUBLIC PreExecutionCheck
VAR_INPUT
    Check : I_PreExecutionChecks;
END_VAR
Check.IsTrue(ipSrcImageX.IsValid, 'ipSrcImageX must contain an image');
Check.IsTrue(ipSrcImageX.IsElementType(ETcVnElementType.TCVN_ET_REAL) OR
             ipSrcImageX.IsElementType(ETcVnElementType.TCVN_ET_LREAL), 'Coordinate images must contain REAL or LREAL elements');
Check.IsTrue(ipSrcImageY.IsValid, 'ipSrcImageY must contain an image');
Check.IsTrue(ImagesHaveMatchingPixelFormats(ipSrcImageX.Value, ipSrcImageY.Value), 'Source images must have matching pixel formats');
Check.IsTrue(IsImage1SizeEqualToImage2Size(ipSrcImageX.Value, ipSrcImageY.Value), 'Source images must have matching dimensions');
END_METHOD

END_FUNCTION_BLOCK

// ---- Nodes/Geometric and Coord Transform/Node_F_VN_ConvertCartesianToPolarMagnitudeImage.TcPOU
{attribute 'linkalways'}
{attribute 'no_explicit_call' := 'This FB is a CLASS and must be accessed using methods or properties'}
{attribute 'enable_dynamic_creation'}
FUNCTION_BLOCK Node_F_VN_ConvertCartesianToPolarMagnitudeImage EXTENDS VisionNode
VAR
    ipSrcImageX : _ITcVnImage;
    ipSrcImageY : _ITcVnImage;
    ipDestImageMag : _ITcVnImage;
    hrPrev : _HRESULT(S_OK);
    hresult : _HRESULT(S_OK);
END_VAR

METHOD PUBLIC Clone : I_Node
VAR
    pNode : POINTER TO Node_F_VN_ConvertCartesianToPolarMagnitudeImage;
END_VAR
pNode := __NEW(Node_F_VN_ConvertCartesianToPolarMagnitudeImage);
Clone := pNode^;
END_METHOD

METHOD FB_init : BOOL
VAR_INPUT
    bInitRetains : BOOL;
    bInCopyCode : BOOL;
END_VAR
AddInput('ipSrcImageX', ipSrcImageX);
AddInput('ipSrcImageY', ipSrcImageY);
AddOutput('ipDestImageMag', ipDestImageMag);
AddInput('hrPrev', hrPrev);
AddOutput('hresult', hresult);
END_METHOD

METHOD PROTECTED OnExecute
hresult.Value := F_VN_ConvertCartesianToPolarMagnitudeImage(
    ipSrcImageX := ipSrcImageX.Value,
    ipSrcImageY := ipSrcImageY.Value,
    ipDestImageMag := ipDestImageMag.Value,
    hrPrev := hrPrev.Value);
END_METHOD

METHOD PUBLIC PreExecutionCheck
VAR_INPUT
    Check : I_PreExecutionChecks;
END_VAR
Check.IsTrue(ipSrcImageX.IsValid, 'ipSrcImageX must contain an image');
Check.IsTrue(ipSrcImageX.IsElementType(ETcVnElementType.TCVN_ET_REAL) OR
             ipSrcImageX.IsElementType(ETcVnElementType.TCVN_ET_LREAL), 'Coordinate images must contain REAL or LREAL elements');
Check.IsTrue(ipSrcImageY.IsValid, 'ipSrcImageY must contain an image');
Check.IsTrue(ImagesHaveMatchingPixelFormats(ipSrcImageX.Value, ipSrcImageY.Value), 'Source images must have matching pixel formats');
Check.IsTrue(IsImage1SizeEqualToImage2Size(ipSrcImageX.Value, ipSrcImageY.Value), 'Source images must have matching dimensions');
END_METHOD

END_FUNCTION_BLOCK

// ---- Nodes/Geometric and Coord Transform/Node_F_VN_ConvertPolarToCartesianImages.TcPOU
{attribute 'linkalways'}
{attribute 'no_explicit_call' := 'This FB is a CLASS and must be accessed using methods or properties'}
{attribute 'enable_dynamic_creation'}
FUNCTION_BLOCK Node_F_VN_ConvertPolarToCartesianImages EXTENDS VisionNode
VAR
    ipSrcImageMag : _ITcVnImage;
    ipSrcImageAng : _ITcVnImage;
    ipDestImageX : _ITcVnImage;
    ipDestImageY : _ITcVnImage;
    hrPrev : _HRESULT(S_OK);
    hresult : _HRESULT(S_OK);
END_VAR

METHOD PUBLIC Clone : I_Node
VAR
    pNode : POINTER TO Node_F_VN_ConvertPolarToCartesianImages;
END_VAR
pNode := __NEW(Node_F_VN_ConvertPolarToCartesianImages);
Clone := pNode^;
END_METHOD

METHOD FB_init : BOOL
VAR_INPUT
    bInitRetains : BOOL;
    bInCopyCode : BOOL;
END_VAR
AddInput('ipSrcImageMag', ipSrcImageMag);
AddInput('ipSrcImageAng', ipSrcImageAng);
AddOutput('ipDestImageX', ipDestImageX);
AddOutput('ipDestImageY', ipDestImageY);
AddInput('hrPrev', hrPrev);
AddOutput('hresult', hresult);
END_METHOD

METHOD PROTECTED OnExecute
hresult.Value := F_VN_ConvertPolarToCartesianImages(
    ipSrcImageMag := ipSrcImageMag.Value,
    ipSrcImageAng := ipSrcImageAng.Value,
    ipDestImageX := ipDestImageX.Value,
    ipDestImageY := ipDestImageY.Value,
    hrPrev := hrPrev.Value);
END_METHOD

METHOD PUBLIC PreExecutionCheck
VAR_INPUT
    Check : I_PreExecutionChecks;
END_VAR
Check.IsTrue(ipSrcImageMag.IsValid, 'ipSrcImageMag must contain an image');
Check.IsTrue(ipSrcImageMag.IsElementType(ETcVnElementType.TCVN_ET_REAL) OR
             ipSrcImageMag.IsElementType(ETcVnElementType.TCVN_ET_LREAL), 'Coordinate images must contain REAL or LREAL elements');
Check.IsTrue(ipSrcImageAng.IsValid, 'ipSrcImageAng must contain an image');
Check.IsTrue(ImagesHaveMatchingPixelFormats(ipSrcImageMag.Value, ipSrcImageAng.Value), 'Source images must have matching pixel formats');
Check.IsTrue(IsImage1SizeEqualToImage2Size(ipSrcImageMag.Value, ipSrcImageAng.Value), 'Source images must have matching dimensions');
END_METHOD

END_FUNCTION_BLOCK

// ---- Nodes/Geometric and Coord Transform/Node_F_VN_ConvertPolarToCartesianImagesExp.TcPOU
{attribute 'linkalways'}
{attribute 'no_explicit_call' := 'This FB is a CLASS and must be accessed using methods or properties'}
{attribute 'enable_dynamic_creation'}
FUNCTION_BLOCK Node_F_VN_ConvertPolarToCartesianImagesExp EXTENDS VisionNode
VAR
    ipSrcImageMag : _ITcVnImage;
    ipSrcImageAng : _ITcVnImage;
    ipDestImageX : _ITcVnImage;
    ipDestImageY : _ITcVnImage;
    bAngleInDegrees : _BOOL(FALSE);
    hrPrev : _HRESULT(S_OK);
    hresult : _HRESULT(S_OK);
END_VAR

METHOD PUBLIC Clone : I_Node
VAR
    pNode : POINTER TO Node_F_VN_ConvertPolarToCartesianImagesExp;
END_VAR
pNode := __NEW(Node_F_VN_ConvertPolarToCartesianImagesExp);
Clone := pNode^;
END_METHOD

METHOD FB_init : BOOL
VAR_INPUT
    bInitRetains : BOOL;
    bInCopyCode : BOOL;
END_VAR
AddInput('ipSrcImageMag', ipSrcImageMag);
AddInput('ipSrcImageAng', ipSrcImageAng);
AddOutput('ipDestImageX', ipDestImageX);
AddOutput('ipDestImageY', ipDestImageY);
AddParameter('bAngleInDegrees', bAngleInDegrees);
AddInput('hrPrev', hrPrev);
AddOutput('hresult', hresult);
END_METHOD

METHOD PROTECTED OnExecute
hresult.Value := F_VN_ConvertPolarToCartesianImagesExp(
    ipSrcImageMag := ipSrcImageMag.Value,
    ipSrcImageAng := ipSrcImageAng.Value,
    ipDestImageX := ipDestImageX.Value,
    ipDestImageY := ipDestImageY.Value,
    bAngleInDegrees := bAngleInDegrees.Value,
    hrPrev := hrPrev.Value);
END_METHOD

METHOD PUBLIC PreExecutionCheck
VAR_INPUT
    Check : I_PreExecutionChecks;
END_VAR
Check.IsTrue(ipSrcImageMag.IsValid, 'ipSrcImageMag must contain an image');
Check.IsTrue(ipSrcImageMag.IsElementType(ETcVnElementType.TCVN_ET_REAL) OR
             ipSrcImageMag.IsElementType(ETcVnElementType.TCVN_ET_LREAL), 'Coordinate images must contain REAL or LREAL elements');
Check.IsTrue(ipSrcImageAng.IsValid, 'ipSrcImageAng must contain an image');
Check.IsTrue(ImagesHaveMatchingPixelFormats(ipSrcImageMag.Value, ipSrcImageAng.Value), 'Source images must have matching pixel formats');
Check.IsTrue(IsImage1SizeEqualToImage2Size(ipSrcImageMag.Value, ipSrcImageAng.Value), 'Source images must have matching dimensions');
END_METHOD

END_FUNCTION_BLOCK

// ---- Nodes/Geometric and Coord Transform/Node_F_VN_ConvertMaps.TcPOU
{attribute 'linkalways'}
{attribute 'no_explicit_call' := 'This FB is a CLASS and must be accessed using methods or properties'}
{attribute 'enable_dynamic_creation'}
FUNCTION_BLOCK Node_F_VN_ConvertMaps EXTENDS VisionNode
VAR
    ipSrcMap1 : _ITcVnImage;
    ipSrcMap2 : _ITcVnImage;
    ipDestMap1 : _ITcVnImage;
    ipDestMap2 : _ITcVnImage;
    eDestMap1Type : _ETcVnElementType(ETcVnElementType.TCVN_ET_INT);
    nDestMap1Channels : _UINT(2);
    hrPrev : _HRESULT(S_OK);
    hresult : _HRESULT(S_OK);
END_VAR

METHOD PUBLIC Clone : I_Node
VAR
    pNode : POINTER TO Node_F_VN_ConvertMaps;
END_VAR
pNode := __NEW(Node_F_VN_ConvertMaps);
Clone := pNode^;
END_METHOD

METHOD FB_init : BOOL
VAR_INPUT
    bInitRetains : BOOL;
    bInCopyCode : BOOL;
END_VAR
AddInput('ipSrcMap1', ipSrcMap1);
AddInput('ipSrcMap2', ipSrcMap2);
AddOutput('ipDestMap1', ipDestMap1);
AddOutput('ipDestMap2', ipDestMap2);
AddParameter('eDestMap1Type', eDestMap1Type);
AddParameter('nDestMap1Channels', nDestMap1Channels);
AddInput('hrPrev', hrPrev);
AddOutput('hresult', hresult);
END_METHOD

METHOD PROTECTED OnExecute
hresult.Value := F_VN_ConvertMaps(
    ipSrcMap1 := ipSrcMap1.Value,
    ipSrcMap2 := ipSrcMap2.Value,
    ipDestMap1 := ipDestMap1.Value,
    ipDestMap2 := ipDestMap2.Value,
    eDestMap1Type := eDestMap1Type.Value,
    nDestMap1Channels := nDestMap1Channels.Value,
    hrPrev := hrPrev.Value);
END_METHOD

METHOD PUBLIC PreExecutionCheck
VAR_INPUT
    Check : I_PreExecutionChecks;
END_VAR
Check.IsTrue(IsRemapMapPairValid(ipSrcMap1.Value, ipSrcMap2.Value), 'Unsupported source map pair: use REAL XY, separate REAL X/Y, or INT XY with optional UINT coefficients');
Check.IsTrue((eDestMap1Type.Value = ETcVnElementType.TCVN_ET_REAL) OR
             (eDestMap1Type.Value = ETcVnElementType.TCVN_ET_INT), 'Destination map type must be REAL or INT');
Check.IsTrue((nDestMap1Channels.Value = 1) OR (nDestMap1Channels.Value = 2), 'Destination map must have 1 or 2 channels');
Check.IsTrue((eDestMap1Type.Value <> ETcVnElementType.TCVN_ET_INT) OR
             (nDestMap1Channels.Value = 2), 'Fixed-point destination map must have 2 channels');
Check.IsTrue((ipDestMap1.Value = 0) OR ((ipDestMap1.Value <> ipSrcMap1.Value) AND (ipDestMap1.Value <> ipSrcMap2.Value)), 'ipDestMap1 must be different from the source maps');
Check.IsTrue((ipDestMap2.Value = 0) OR ((ipDestMap2.Value <> ipSrcMap1.Value) AND (ipDestMap2.Value <> ipSrcMap2.Value)), 'ipDestMap2 must be different from the source maps');
Check.IsTrue((ipDestMap1.Value = 0) OR (ipDestMap1.Value <> ipDestMap2.Value), 'Destination maps must be different images');
END_METHOD

END_FUNCTION_BLOCK

// ---- Functions/Checks/IsRemapMapPairValid.TcPOU
FUNCTION IsRemapMapPairValid : BOOL
VAR_INPUT
    Map1 : ITcVnImage;
    Map2 : ITcVnImage;
END_VAR
VAR
    format1 : TcVnPixelFormat;
    format2 : TcVnPixelFormat;
    map1IsReal : BOOL;
    map1IsInt : BOOL;
END_VAR

// The map pair determines the destination size; it need not match the source image size.
IF NOT IsValidImage(Map1) THEN
    RETURN;
END_IF
IF FAILED(Map1.GetPixelFormat(format1)) THEN
    RETURN;
END_IF
map1IsReal := ImageHasElementType(Map1, ETcVnElementType.TCVN_ET_REAL);
map1IsInt := ImageHasElementType(Map1, ETcVnElementType.TCVN_ET_INT);

IF Map2 = 0 THEN
    // Interleaved floating-point coordinates, or rounded fixed-point coordinates.
    IsRemapMapPairValid := (format1.nChannels = 2) AND (map1IsReal OR map1IsInt);
    RETURN;
END_IF
IF FAILED(Map2.GetPixelFormat(format2)) THEN
    RETURN;
END_IF
IF NOT IsImage1SizeEqualToImage2Size(Map1, Map2) THEN
    RETURN;
END_IF
IF format2.nChannels <> 1 THEN
    RETURN;
END_IF
// Separate floating-point X/Y maps, or fixed-point coordinates plus interpolation coefficients.
IsRemapMapPairValid := ((format1.nChannels = 1) AND map1IsReal AND
                       ImageHasElementType(Map2, ETcVnElementType.TCVN_ET_REAL)) OR
                      ((format1.nChannels = 2) AND map1IsInt AND
                       ImageHasElementType(Map2, ETcVnElementType.TCVN_ET_UINT));

END_FUNCTION

// ---- Nodes/Geometric and Coord Transform/Node_F_VN_RemapImage.TcPOU
{attribute 'linkalways'}
{attribute 'no_explicit_call' := 'This FB is a CLASS and must be accessed using methods or properties'}
{attribute 'enable_dynamic_creation'}
FUNCTION_BLOCK Node_F_VN_RemapImage EXTENDS VisionNode
VAR
    ipSrcImage : _ITcVnImage;
    ipDestImage : _ITcVnImage;
    ipMap1 : _ITcVnImage;
    ipMap2 : _ITcVnImage;
    hrPrev : _HRESULT(S_OK);
    hresult : _HRESULT(S_OK);
END_VAR

METHOD PUBLIC Clone : I_Node
VAR
    pNode : POINTER TO Node_F_VN_RemapImage;
END_VAR
pNode := __NEW(Node_F_VN_RemapImage);
Clone := pNode^;
END_METHOD

METHOD FB_init : BOOL
VAR_INPUT
    bInitRetains : BOOL;
    bInCopyCode : BOOL;
END_VAR
AddInput('ipSrcImage', ipSrcImage);
AddOutput('ipDestImage', ipDestImage);
AddInput('ipMap1', ipMap1);
AddInput('ipMap2', ipMap2);
AddInput('hrPrev', hrPrev);
AddOutput('hresult', hresult);
END_METHOD

METHOD PROTECTED OnExecute
hresult.Value := F_VN_RemapImage(
    ipSrcImage := ipSrcImage.Value,
    ipDestImage := ipDestImage.Value,
    ipMap1 := ipMap1.Value,
    ipMap2 := ipMap2.Value,
    hrPrev := hrPrev.Value);
END_METHOD

METHOD PUBLIC PreExecutionCheck
VAR_INPUT
    Check : I_PreExecutionChecks;
END_VAR
Check.IsTrue(ipSrcImage.IsValid, 'ipSrcImage must contain an image');
Check.IsTrue((ipDestImage.Value = 0) OR (ipDestImage.Value <> ipSrcImage.Value), 'Destination must be different from the source image');
Check.IsTrue(IsRemapMapPairValid(ipMap1.Value, ipMap2.Value), 'Unsupported remap pair: use REAL XY, separate REAL X/Y, or INT XY with optional UINT coefficients');
END_METHOD

END_FUNCTION_BLOCK

// ---- Nodes/Geometric and Coord Transform/Node_F_VN_RemapImageExp.TcPOU
{attribute 'linkalways'}
{attribute 'no_explicit_call' := 'This FB is a CLASS and must be accessed using methods or properties'}
{attribute 'enable_dynamic_creation'}
FUNCTION_BLOCK Node_F_VN_RemapImageExp EXTENDS VisionNode
VAR
    ipSrcImage : _ITcVnImage;
    ipDestImage : _ITcVnImage;
    ipMap1 : _ITcVnImage;
    ipMap2 : _ITcVnImage;
    bRelativeMap : _BOOL(FALSE);
    eInterpolationType : _ETcVnInterpolationType(ETcVnInterpolationType.TCVN_IT_BILINEAR);
    eBorderInterpolation : _ETcVnBorderInterpolationMethod(ETcVnBorderInterpolationMethod.TCVN_BIM_CONSTANT);
    aBorderValue : _TcVnVector4_LREAL;
    hrPrev : _HRESULT(S_OK);
    hresult : _HRESULT(S_OK);
END_VAR

METHOD PUBLIC Clone : I_Node
VAR
    pNode : POINTER TO Node_F_VN_RemapImageExp;
END_VAR
pNode := __NEW(Node_F_VN_RemapImageExp);
Clone := pNode^;
END_METHOD

METHOD FB_init : BOOL
VAR_INPUT
    bInitRetains : BOOL;
    bInCopyCode : BOOL;
END_VAR
AddInput('ipSrcImage', ipSrcImage);
AddOutput('ipDestImage', ipDestImage);
AddInput('ipMap1', ipMap1);
AddInput('ipMap2', ipMap2);
AddParameter('bRelativeMap', bRelativeMap);
AddParameter('eInterpolationType', eInterpolationType);
AddParameter('eBorderInterpolation', eBorderInterpolation);
AddInput('aBorderValue', aBorderValue);
AddInput('hrPrev', hrPrev);
AddOutput('hresult', hresult);
END_METHOD

METHOD PROTECTED OnExecute
hresult.Value := F_VN_RemapImageExp(
    ipSrcImage := ipSrcImage.Value,
    ipDestImage := ipDestImage.Value,
    ipMap1 := ipMap1.Value,
    ipMap2 := ipMap2.Value,
    bRelativeMap := bRelativeMap.Value,
    eInterpolationType := eInterpolationType.Value,
    eBorderInterpolation := eBorderInterpolation.Value,
    aBorderValue := aBorderValue.Value,
    hrPrev := hrPrev.Value);
END_METHOD

METHOD PUBLIC PreExecutionCheck
VAR_INPUT
    Check : I_PreExecutionChecks;
END_VAR
Check.IsTrue(ipSrcImage.IsValid, 'ipSrcImage must contain an image');
Check.IsTrue((ipDestImage.Value = 0) OR (ipDestImage.Value <> ipSrcImage.Value), 'Destination must be different from the source image');
Check.IsTrue(IsRemapMapPairValid(ipMap1.Value, ipMap2.Value), 'Unsupported remap pair: use REAL XY, separate REAL X/Y, or INT XY with optional UINT coefficients');
Check.IsTrue((eInterpolationType.Value = ETcVnInterpolationType.TCVN_IT_NEAREST_NEIGHBOR) OR
             (eInterpolationType.Value = ETcVnInterpolationType.TCVN_IT_BILINEAR) OR
             (eInterpolationType.Value = ETcVnInterpolationType.TCVN_IT_BICUBIC) OR
             (eInterpolationType.Value = ETcVnInterpolationType.TCVN_IT_LANCZOS4), 'Unsupported eInterpolationType');
Check.IsTrue((eBorderInterpolation.Value = ETcVnBorderInterpolationMethod.TCVN_BIM_CONSTANT) OR
             (eBorderInterpolation.Value = ETcVnBorderInterpolationMethod.TCVN_BIM_REPLICATE) OR
             (eBorderInterpolation.Value = ETcVnBorderInterpolationMethod.TCVN_BIM_REFLECT) OR
             (eBorderInterpolation.Value = ETcVnBorderInterpolationMethod.TCVN_BIM_WRAP) OR
             (eBorderInterpolation.Value = ETcVnBorderInterpolationMethod.TCVN_BIM_REFLECT_101) OR
             (eBorderInterpolation.Value = ETcVnBorderInterpolationMethod.TCVN_BIM_DEFAULT) OR
             (eBorderInterpolation.Value = ETcVnBorderInterpolationMethod.TCVN_BIM_TRANSPARENT), 'Unsupported eBorderInterpolation');
END_METHOD

END_FUNCTION_BLOCK

// ---- Nodes/Geometric and Coord Transform/Node_F_VN_RemapImageToLogPolarSpaceExp.TcPOU
{attribute 'linkalways'}
{attribute 'no_explicit_call' := 'This FB is a CLASS and must be accessed using methods or properties'}
{attribute 'enable_dynamic_creation'}
FUNCTION_BLOCK Node_F_VN_RemapImageToLogPolarSpaceExp EXTENDS VisionNode
VAR
    ipSrcImage : _ITcVnImage;
    ipDestImage : _ITcVnImage;
    aCenter : _TcVnPoint2_REAL;
    fScale : _LREAL(0);
    eInterpolationType : _ETcVnInterpolationType(ETcVnInterpolationType.TCVN_IT_BILINEAR);
    hrPrev : _HRESULT(S_OK);
    hresult : _HRESULT(S_OK);
END_VAR

METHOD PUBLIC Clone : I_Node
VAR
    pNode : POINTER TO Node_F_VN_RemapImageToLogPolarSpaceExp;
END_VAR
pNode := __NEW(Node_F_VN_RemapImageToLogPolarSpaceExp);
Clone := pNode^;
END_METHOD

METHOD FB_init : BOOL
VAR_INPUT
    bInitRetains : BOOL;
    bInCopyCode : BOOL;
END_VAR
AddInput('ipSrcImage', ipSrcImage);
AddOutput('ipDestImage', ipDestImage);
AddInput('aCenter', aCenter);
AddParameter('fScale', fScale);
AddParameter('eInterpolationType', eInterpolationType);
AddInput('hrPrev', hrPrev);
AddOutput('hresult', hresult);
END_METHOD

METHOD PROTECTED OnExecute
hresult.Value := F_VN_RemapImageToLogPolarSpaceExp(
    ipSrcImage := ipSrcImage.Value,
    ipDestImage := ipDestImage.Value,
    aCenter := aCenter.Value,
    fScale := fScale.Value,
    eInterpolationType := eInterpolationType.Value,
    hrPrev := hrPrev.Value);
END_METHOD

METHOD PUBLIC PreExecutionCheck
VAR_INPUT
    Check : I_PreExecutionChecks;
END_VAR
Check.IsTrue(ipSrcImage.IsValid, 'ipSrcImage must contain an image');
Check.IsTrue((ipDestImage.Value = 0) OR (ipDestImage.Value <> ipSrcImage.Value), 'Destination must be different from the source image');
Check.IsTrue((eInterpolationType.Value = ETcVnInterpolationType.TCVN_IT_NEAREST_NEIGHBOR) OR
             (eInterpolationType.Value = ETcVnInterpolationType.TCVN_IT_BILINEAR) OR
             (eInterpolationType.Value = ETcVnInterpolationType.TCVN_IT_BICUBIC) OR
             (eInterpolationType.Value = ETcVnInterpolationType.TCVN_IT_AREA_BASED) OR
             (eInterpolationType.Value = ETcVnInterpolationType.TCVN_IT_LANCZOS4), 'Unsupported eInterpolationType');
END_METHOD

END_FUNCTION_BLOCK

// ---- Nodes/Geometric and Coord Transform/Node_F_VN_RemapImageToLogPolarSpaceExp2.TcPOU
{attribute 'linkalways'}
{attribute 'no_explicit_call' := 'This FB is a CLASS and must be accessed using methods or properties'}
{attribute 'enable_dynamic_creation'}
FUNCTION_BLOCK Node_F_VN_RemapImageToLogPolarSpaceExp2 EXTENDS VisionNode
VAR
    ipSrcImage : _ITcVnImage;
    ipDestImage : _ITcVnImage;
    aCenter : _TcVnPoint2_REAL;
    fScale : _LREAL(0);
    eInterpolationType : _ETcVnInterpolationType(ETcVnInterpolationType.TCVN_IT_BILINEAR);
    nDestWidth : _DINT(-1);
    nDestHeight : _DINT(-1);
    hrPrev : _HRESULT(S_OK);
    hresult : _HRESULT(S_OK);
END_VAR

METHOD PUBLIC Clone : I_Node
VAR
    pNode : POINTER TO Node_F_VN_RemapImageToLogPolarSpaceExp2;
END_VAR
pNode := __NEW(Node_F_VN_RemapImageToLogPolarSpaceExp2);
Clone := pNode^;
END_METHOD

METHOD FB_init : BOOL
VAR_INPUT
    bInitRetains : BOOL;
    bInCopyCode : BOOL;
END_VAR
AddInput('ipSrcImage', ipSrcImage);
AddOutput('ipDestImage', ipDestImage);
AddInput('aCenter', aCenter);
AddParameter('fScale', fScale);
AddParameter('eInterpolationType', eInterpolationType);
AddParameter('nDestWidth', nDestWidth);
AddParameter('nDestHeight', nDestHeight);
AddInput('hrPrev', hrPrev);
AddOutput('hresult', hresult);
END_METHOD

METHOD PROTECTED OnExecute
hresult.Value := F_VN_RemapImageToLogPolarSpaceExp2(
    ipSrcImage := ipSrcImage.Value,
    ipDestImage := ipDestImage.Value,
    aCenter := aCenter.Value,
    fScale := fScale.Value,
    eInterpolationType := eInterpolationType.Value,
    nDestWidth := nDestWidth.Value,
    nDestHeight := nDestHeight.Value,
    hrPrev := hrPrev.Value);
END_METHOD

METHOD PUBLIC PreExecutionCheck
VAR_INPUT
    Check : I_PreExecutionChecks;
END_VAR
Check.IsTrue(ipSrcImage.IsValid, 'ipSrcImage must contain an image');
Check.IsTrue((ipDestImage.Value = 0) OR (ipDestImage.Value <> ipSrcImage.Value), 'Destination must be different from the source image');
Check.IsTrue((eInterpolationType.Value = ETcVnInterpolationType.TCVN_IT_NEAREST_NEIGHBOR) OR
             (eInterpolationType.Value = ETcVnInterpolationType.TCVN_IT_BILINEAR) OR
             (eInterpolationType.Value = ETcVnInterpolationType.TCVN_IT_BICUBIC) OR
             (eInterpolationType.Value = ETcVnInterpolationType.TCVN_IT_AREA_BASED) OR
             (eInterpolationType.Value = ETcVnInterpolationType.TCVN_IT_LANCZOS4), 'Unsupported eInterpolationType');
Check.IsTrue(nDestWidth.Value >= -1, 'Destination width must be -1 for source width, 0 for automatic, or positive');
Check.IsTrue(nDestHeight.Value >= -1, 'Destination height must be -1 for source height, 0 for automatic, or positive');
END_METHOD

END_FUNCTION_BLOCK

// ---- Nodes/Geometric and Coord Transform/Node_F_VN_RemapImageToPolarSpaceExp.TcPOU
{attribute 'linkalways'}
{attribute 'no_explicit_call' := 'This FB is a CLASS and must be accessed using methods or properties'}
{attribute 'enable_dynamic_creation'}
FUNCTION_BLOCK Node_F_VN_RemapImageToPolarSpaceExp EXTENDS VisionNode
VAR
    ipSrcImage : _ITcVnImage;
    ipDestImage : _ITcVnImage;
    aCenter : _TcVnPoint2_REAL;
    fMaxRadius : _LREAL(0);
    eInterpolationType : _ETcVnInterpolationType(ETcVnInterpolationType.TCVN_IT_BILINEAR);
    hrPrev : _HRESULT(S_OK);
    hresult : _HRESULT(S_OK);
END_VAR

METHOD PUBLIC Clone : I_Node
VAR
    pNode : POINTER TO Node_F_VN_RemapImageToPolarSpaceExp;
END_VAR
pNode := __NEW(Node_F_VN_RemapImageToPolarSpaceExp);
Clone := pNode^;
END_METHOD

METHOD FB_init : BOOL
VAR_INPUT
    bInitRetains : BOOL;
    bInCopyCode : BOOL;
END_VAR
AddInput('ipSrcImage', ipSrcImage);
AddOutput('ipDestImage', ipDestImage);
AddInput('aCenter', aCenter);
AddParameter('fMaxRadius', fMaxRadius);
AddParameter('eInterpolationType', eInterpolationType);
AddInput('hrPrev', hrPrev);
AddOutput('hresult', hresult);
END_METHOD

METHOD PROTECTED OnExecute
hresult.Value := F_VN_RemapImageToPolarSpaceExp(
    ipSrcImage := ipSrcImage.Value,
    ipDestImage := ipDestImage.Value,
    aCenter := aCenter.Value,
    fMaxRadius := fMaxRadius.Value,
    eInterpolationType := eInterpolationType.Value,
    hrPrev := hrPrev.Value);
END_METHOD

METHOD PUBLIC PreExecutionCheck
VAR_INPUT
    Check : I_PreExecutionChecks;
END_VAR
Check.IsTrue(ipSrcImage.IsValid, 'ipSrcImage must contain an image');
Check.IsTrue((ipDestImage.Value = 0) OR (ipDestImage.Value <> ipSrcImage.Value), 'Destination must be different from the source image');
Check.IsTrue((eInterpolationType.Value = ETcVnInterpolationType.TCVN_IT_NEAREST_NEIGHBOR) OR
             (eInterpolationType.Value = ETcVnInterpolationType.TCVN_IT_BILINEAR) OR
             (eInterpolationType.Value = ETcVnInterpolationType.TCVN_IT_BICUBIC) OR
             (eInterpolationType.Value = ETcVnInterpolationType.TCVN_IT_AREA_BASED) OR
             (eInterpolationType.Value = ETcVnInterpolationType.TCVN_IT_LANCZOS4), 'Unsupported eInterpolationType');
Check.IsTrue(fMaxRadius.Value >= 0.0, 'Maximum radius must be non-negative; zero selects it automatically');
END_METHOD

END_FUNCTION_BLOCK

// ---- Nodes/Geometric and Coord Transform/Node_F_VN_RemapImageToPolarSpaceExp2.TcPOU
{attribute 'linkalways'}
{attribute 'no_explicit_call' := 'This FB is a CLASS and must be accessed using methods or properties'}
{attribute 'enable_dynamic_creation'}
FUNCTION_BLOCK Node_F_VN_RemapImageToPolarSpaceExp2 EXTENDS VisionNode
VAR
    ipSrcImage : _ITcVnImage;
    ipDestImage : _ITcVnImage;
    aCenter : _TcVnPoint2_REAL;
    fMaxRadius : _LREAL(0);
    eInterpolationType : _ETcVnInterpolationType(ETcVnInterpolationType.TCVN_IT_BILINEAR);
    nDestWidth : _DINT(-1);
    nDestHeight : _DINT(-1);
    hrPrev : _HRESULT(S_OK);
    hresult : _HRESULT(S_OK);
END_VAR

METHOD PUBLIC Clone : I_Node
VAR
    pNode : POINTER TO Node_F_VN_RemapImageToPolarSpaceExp2;
END_VAR
pNode := __NEW(Node_F_VN_RemapImageToPolarSpaceExp2);
Clone := pNode^;
END_METHOD

METHOD FB_init : BOOL
VAR_INPUT
    bInitRetains : BOOL;
    bInCopyCode : BOOL;
END_VAR
AddInput('ipSrcImage', ipSrcImage);
AddOutput('ipDestImage', ipDestImage);
AddInput('aCenter', aCenter);
AddParameter('fMaxRadius', fMaxRadius);
AddParameter('eInterpolationType', eInterpolationType);
AddParameter('nDestWidth', nDestWidth);
AddParameter('nDestHeight', nDestHeight);
AddInput('hrPrev', hrPrev);
AddOutput('hresult', hresult);
END_METHOD

METHOD PROTECTED OnExecute
hresult.Value := F_VN_RemapImageToPolarSpaceExp2(
    ipSrcImage := ipSrcImage.Value,
    ipDestImage := ipDestImage.Value,
    aCenter := aCenter.Value,
    fMaxRadius := fMaxRadius.Value,
    eInterpolationType := eInterpolationType.Value,
    nDestWidth := nDestWidth.Value,
    nDestHeight := nDestHeight.Value,
    hrPrev := hrPrev.Value);
END_METHOD

METHOD PUBLIC PreExecutionCheck
VAR_INPUT
    Check : I_PreExecutionChecks;
END_VAR
Check.IsTrue(ipSrcImage.IsValid, 'ipSrcImage must contain an image');
Check.IsTrue((ipDestImage.Value = 0) OR (ipDestImage.Value <> ipSrcImage.Value), 'Destination must be different from the source image');
Check.IsTrue((eInterpolationType.Value = ETcVnInterpolationType.TCVN_IT_NEAREST_NEIGHBOR) OR
             (eInterpolationType.Value = ETcVnInterpolationType.TCVN_IT_BILINEAR) OR
             (eInterpolationType.Value = ETcVnInterpolationType.TCVN_IT_BICUBIC) OR
             (eInterpolationType.Value = ETcVnInterpolationType.TCVN_IT_AREA_BASED) OR
             (eInterpolationType.Value = ETcVnInterpolationType.TCVN_IT_LANCZOS4), 'Unsupported eInterpolationType');
Check.IsTrue(fMaxRadius.Value >= 0.0, 'Maximum radius must be non-negative; zero selects it automatically');
Check.IsTrue(nDestWidth.Value >= -1, 'Destination width must be -1 for source width, 0 for automatic, or positive');
Check.IsTrue(nDestHeight.Value >= -1, 'Destination height must be -1 for source height, 0 for automatic, or positive');
END_METHOD

END_FUNCTION_BLOCK

// ---- Nodes/Image Color and Contrast Processing/Node_F_VN_InvertImageColorExp.TcPOU
{attribute 'linkalways'}
{attribute 'no_explicit_call' := 'This FB is a CLASS and must be accessed using methods or properties'}
{attribute 'enable_dynamic_creation'}
FUNCTION_BLOCK Node_F_VN_InvertImageColorExp EXTENDS VisionNode
VAR
    ipSrcImage : _ITcVnImage;
    ipDestImage : _ITcVnImage;
    fMaxValue : _LREAL(-1);
    hrPrev : _HRESULT(S_OK);
    hresult : _HRESULT(S_OK);
END_VAR

METHOD PUBLIC Clone : I_Node
VAR
    pNode : POINTER TO Node_F_VN_InvertImageColorExp;
END_VAR
pNode := __NEW(Node_F_VN_InvertImageColorExp);
Clone := pNode^;
END_METHOD

METHOD FB_init : BOOL
VAR_INPUT
    bInitRetains : BOOL;
    bInCopyCode : BOOL;
END_VAR
AddInput('ipSrcImage', ipSrcImage);
AddOutput('ipDestImage', ipDestImage);
AddParameter('fMaxValue', fMaxValue);
AddInput('hrPrev', hrPrev);
AddOutput('hresult', hresult);
END_METHOD

METHOD PROTECTED OnExecute
hresult.Value := F_VN_InvertImageColorExp(
    ipSrcImage := ipSrcImage.Value,
    ipDestImage := ipDestImage.Value,
    fMaxValue := fMaxValue.Value,
    hrPrev := hrPrev.Value);
END_METHOD

METHOD PUBLIC PreExecutionCheck
VAR_INPUT
    Check : I_PreExecutionChecks;
END_VAR
Check.IsTrue(ipSrcImage.IsValid, 'ipSrcImage must contain an image');
END_METHOD

END_FUNCTION_BLOCK

// ---- Nodes/Image Color and Contrast Processing/Node_F_VN_NormalizeImageExp.TcPOU
{attribute 'linkalways'}
{attribute 'no_explicit_call' := 'This FB is a CLASS and must be accessed using methods or properties'}
{attribute 'enable_dynamic_creation'}
FUNCTION_BLOCK Node_F_VN_NormalizeImageExp EXTENDS VisionNode
VAR
    ipSrcImage : _ITcVnImage;
    ipDestImage : _ITcVnImage;
    fAlpha : _LREAL(0);
    fBeta : _LREAL(255);
    eNormType : _ETcVnNormalizationType(ETcVnNormalizationType.TCVN_NT_MINMAX);
    eDestType : _ETcVnElementType(ETcVnElementType.TCVN_ET_SAME_AS_SOURCE);
    ipMask : _ITcVnImage;
    hrPrev : _HRESULT(S_OK);
    hresult : _HRESULT(S_OK);
END_VAR

METHOD PUBLIC Clone : I_Node
VAR
    pNode : POINTER TO Node_F_VN_NormalizeImageExp;
END_VAR
pNode := __NEW(Node_F_VN_NormalizeImageExp);
Clone := pNode^;
END_METHOD

METHOD FB_init : BOOL
VAR_INPUT
    bInitRetains : BOOL;
    bInCopyCode : BOOL;
END_VAR
AddInput('ipSrcImage', ipSrcImage);
AddOutput('ipDestImage', ipDestImage);
AddParameter('fAlpha', fAlpha);
AddParameter('fBeta', fBeta);
AddParameter('eNormType', eNormType);
AddParameter('eDestType', eDestType);
AddInput('ipMask', ipMask);
AddInput('hrPrev', hrPrev);
AddOutput('hresult', hresult);
END_METHOD

METHOD PROTECTED OnExecute
hresult.Value := F_VN_NormalizeImageExp(
    ipSrcImage := ipSrcImage.Value,
    ipDestImage := ipDestImage.Value,
    fAlpha := fAlpha.Value,
    fBeta := fBeta.Value,
    eNormType := eNormType.Value,
    eDestType := eDestType.Value,
    ipMask := ipMask.Value,
    hrPrev := hrPrev.Value);
END_METHOD

METHOD PUBLIC PreExecutionCheck
VAR_INPUT
    Check : I_PreExecutionChecks;
END_VAR
Check.IsTrue(ipSrcImage.IsValid, 'ipSrcImage must contain an image');
IF ipMask.Value <> 0 THEN
    Check.IsTrue(ipMask.IsValid, 'ipMask must contain an image when connected');
    Check.IsTrue(IsImage1SizeEqualToImage2Size(ipSrcImage.Value, ipMask.Value), 'Source and mask must have matching dimensions');
END_IF
Check.IsTrue((eNormType.Value = ETcVnNormalizationType.TCVN_NT_INF) OR
             (eNormType.Value = ETcVnNormalizationType.TCVN_NT_L1) OR
             (eNormType.Value = ETcVnNormalizationType.TCVN_NT_L2) OR
             (eNormType.Value = ETcVnNormalizationType.TCVN_NT_MINMAX), 'Unsupported eNormType');
END_METHOD

END_FUNCTION_BLOCK

// ---- VisionPack.TcPOU
{attribute 'linkalways'} 
{attribute 'no_explicit_call' := 'This FB is a CLASS and must be accessed using methods or properties'}
{attribute 'enable_dynamic_creation'}
FUNCTION_BLOCK VisionPack IMPLEMENTS I_GraphPack
VAR
	visionDatatypePack : VisionDatatypePack;
	visionNodePack : VisionNodePack;
END_VAR

METHOD Register
VAR_INPUT
	Datatypes : I_Datatypes;
	NodeFactory : I_NodeFactory;
END_VAR
visionDatatypePack.RegisterWithDatatypes(Datatypes);
visionNodePack.RegisterWithNodeFactory(NodeFactory);
END_METHOD

END_FUNCTION_BLOCK
